(* CODESYS project INICIANDO.project

Project tree, tasks and I/O mapping:
  Device : CODESYS Control Win V3, 3S - Smart Software Solutions GmbH, order no. 305021, version 3.5.11.30
    application Application
      libraries: Standard, * (System)
      task MainTask (cyclic, interval t#20ms, priority 1) calls PLC_PRG
      task VISU_TASK (cyclic, interval 100 ms, priority 31) calls VisuElems.Visu_Prg
      program PLC_PRG [LD]
      visualisation Visualization
  libraries: VisuSymbols, 3.5.10.0 (System)
  text list GlobalTextList
*)

// Device/Application/PLC_PRG
PROGRAM PLC_PRG
VAR
	B1 : BOOL;
	B2 : BOOL;
	S1 : BOOL;
	B3: BOOL;
END_VAR

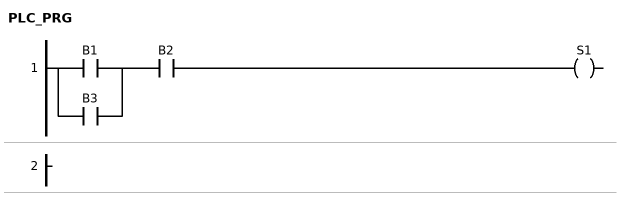
// NETWORK 1
S1 := (B1 OR B3) AND B2;

// NETWORK 2

END_PROGRAM

// Device/Application/Visualization
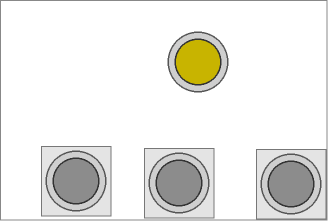
VISUALIZATION Visualization  // 328x221
    Lamp1 (163,27 70x70), variable: PLC_PRG.S1, style: Lamp-Lamp1-Yellow
    PushSwitch (41,146 70x70), variable: PLC_PRG.B1, behaviour: TOGGLE, style: Switch-PushSwitch-Gray
    PushSwitch (144,148 70x70), variable: PLC_PRG.B2, behaviour: TOGGLE, style: Switch-PushSwitch-Gray
    PushSwitch (256,149 70x70), variable: PLC_PRG.B3, behaviour: TOGGLE, style: Switch-PushSwitch-Gray
END_VISUALIZATION
